    string sName = "NetOut46"
  [NetOut47]
    bool bActive
    bool bEnable = true
    dio dDio = {link=ApplicomIO-1\TOPIC1_A-BLOCKA\%Q47}
    string sID = "NetOut47"
    string sName = "NetOut47"
  [NetOut48]
    bool bActive
    bool bEnable = true
    dio dDio = {link=ApplicomIO-1\TOPIC1_A-BLOCKA\%Q48}
    string sID = "NetOut48"
    string sName = "NetOut48"
  [NetOut49]
    bool bActive
    bool bEnable = true
    dio dDio = {link=ApplicomIO-1\TOPIC1_A-BLOCKA\%Q49}
    string sID = "NetOut49"
    string sName = "NetOut49"
  [NetOut50]
    bool bActive
    bool bEnable = true
    dio dDio = {link=ApplicomIO-1\TOPIC1_A-BLOCKA\%Q50}
    string sID = "NetOut50"
    string sName = "NetOut50"
  [NetOut51]
    bool bActive
    bool bEnable = true
    dio dDio = {link=ApplicomIO-1\TOPIC1_A-BLOCKA\%Q51}
    string sID = "NetOut51"
    string sName = "NetOut51"
  [NetOut52]
    bool bActive
    bool bEnable = true
    dio dDio = {link=ApplicomIO-1\TOPIC1_A-BLOCKA\%Q52}
    string sID = "NetOut52"
    string sName = "NetOut52"
  [NetOut53]
    bool bActive
    bool bEnable = true
    dio dDio = {link=ApplicomIO-1\TOPIC1_A-BLOCKA\%Q53}
    string sID = "NetOut53"
    string sName = "NetOut53"
  [NetOut54]
    bool bActive
    bool bEnable = true
    dio dDio = {link=ApplicomIO-1\TOPIC1_A-BLOCKA\%Q54}
    string sID = "NetOut54"
    string sName = "NetOut54"
  [NetOut55]
    bool bActive
    bool bEnable = true
    dio dDio = {link=ApplicomIO-1\TOPIC1_A-BLOCKA\%Q55}
    string sID = "NetOut55"
    string sName = "NetOut55"
  [NetOut56]
    bool bActive
    bool bEnable = true
    dio dDio = {link=ApplicomIO-1\TOPIC1_A-BLOCKA\%Q56}
    string sID = "NetOut56"
    string sName = "NetOut56"
  [NetOut57]
    bool bActive
    bool bEnable = true
    dio dDio = {link=ApplicomIO-1\TOPIC1_A-BLOCKA\%Q57}
    string sID = "NetOut57"
    string sName = "NetOut57"
  [NetOut58]
    bool bActive
    bool bEnable = true
    dio dDio = {link=ApplicomIO-1\TOPIC1_A-BLOCKA\%Q58}
    string sID = "NetOut58"
    string sName = "NetOut58"
  [NetOut59]
    bool bActive
    bool bEnable = true
    dio dDio = {link=ApplicomIO-1\TOPIC1_A-BLOCKA\%Q59}
    string sID = "NetOut59"
    string sName = "NetOut59"
  [NetOut60]
    bool bActive
    bool bEnable = true
    dio dDio = {link=ApplicomIO-1\TOPIC1_A-BLOCKA\%Q60}
    string sID = "NetOut60"
    string sName = "NetOut60"
  [NetOut61]
    bool bActive
    bool bEnable = true
    dio dDio = {link=ApplicomIO-1\TOPIC1_A-BLOCKA\%Q61}
    string sID = "NetOut61"
    string sName = "NetOut61"
  [NetOut62]
    bool bActive
    bool bEnable = true
    dio dDio = {link=ApplicomIO-1\TOPIC1_A-BLOCKA\%Q62}
    string sID = "NetOut62"
    string sName = "NetOut62"
  [NetOut63]
    bool bActive
    bool bEnable = true
    dio dDio = {link=ApplicomIO-1\TOPIC1_A-BLOCKA\%Q63}
    string sID = "NetOut63"
    string sName = "NetOut63"
  [fOut0]
    bool bActive = true
    bool bEnable = true
    dio dDio = {link=fOut0}
    string sID = "fOut0"
    string sName = "fOut0"
  [valve1]
    bool bActive = true
    bool bEnable = true
    dio dDio = {link=valve1}
    string sID = "valve1"
    string sName = "valve1"
  [valve2]
    bool bActive = true
    bool bEnable = true
    dio dDio = {link=valve2}
    string sID = "valve2"
    string sName = "valve2"
public num nCounter[10]
public string sCondition[6]
  [0] = "!="
  [1] = ">="
  [2] = "> "
  [3] = "< "
  [4] = "<="
  [5] = "=="
public string sOperator[4]
  [0] = "= "
  [1] = "=NUM "
  [2] = "+1"
  [3] = "-1"

--- decompose_num.pgx ---
public program decompose_num(string& x_sItem[] (dimensions=1), string& x_sName (dimensions=1), num& x_nOperator (dimensions=1), num& x_nValue (dimensions=1))
  local num i
  local num l_nPos
  local num l_nSize
  local string l_sItem
  local bool l_bOk
  local string l_sItem2
begin
  //
  // decompose into Index-Operator-Value-Mode
  //
  for i=0 to size(sOperator)-1
    // Operator
    l_nPos=find(x_sItem,sOperator[i])
    if l_nPos!=-1
      x_nOperator=i
      i=size(sOperator)-1
    endIf
  endFor
  if l_nPos!=-1
    // find the Index
    call getSize_num(l_nSize)
    for i=0 to l_nSize-1
      // search it
      call get_num(l_sItem,i)
      if l_sItem==left(x_sItem,l_nPos)
        x_sName=l_sItem
        i=l_nSize-1
      endIf
    endFor
    // get the value
    if x_nOperator==1
      // found the value
      l_sItem2=right(x_sItem,len(x_sItem)-l_nPos-len(sOperator[1]))
      if size(x_sItem)>1
        x_sItem[1]=l_sItem
      endIf
      for i=0 to l_nSize-1
        // search it
        call get_num(l_sItem,i)
        if l_sItem==l_sItem2
          call getValue_num(x_nValue,l_sItem)
          return
        endIf
      endFor
    else
      toNum(right(x_sItem,len(x_sItem)-l_nPos-2),x_nValue,l_bOk)
    endIf
  else
    x_sName=""
  endIf
end

--- decompose_wait.pgx ---
public program decompose_wait(string& x_sItem[] (dimensions=1), string& x_sName (dimensions=1), num& x_nOperator (dimensions=1), num& x_nValue (dimensions=1))
  local num i
  local num l_nPos
  local num l_nSize
  local string l_sItem
  local bool l_bOk
  local string l_sItem2
begin
  //
  // decompose into Index-Operator-Value-Mode
  //
  for i=0 to size(sCondition)-1
    // Operator
    l_nPos=find(x_sItem,sCondition[i])
    if l_nPos!=-1
      x_nOperator=i
      i=size(sCondition)-1
    endIf
  endFor
  if l_nPos!=-1
    // find the Index
    call getSize_num(l_nSize)
    for i=0 to l_nSize-1
      // search it
      call get_num(l_sItem,i)
      if l_sItem==left(x_sItem,l_nPos)
        x_sName=l_sItem
        i=l_nSize-1
      endIf
    endFor
    // get the value
    toNum(right(x_sItem,len(x_sItem)-l_nPos-2),x_nValue,l_bOk)
    if !l_bOk
      // found the value
      l_sItem2=right(x_sItem,len(x_sItem)-l_nPos-len(sCondition[1]))
      if size(x_sItem)>1
        x_sItem[1]=l_sItem
      endIf
      for i=0 to l_nSize-1
        // search it
        call get_num(l_sItem,i)
        if l_sItem==l_sItem2
          call getValue_num(x_nValue,l_sItem)
          return
        endIf
      endFor
    endIf
  else
    x_sName=""
  endIf
end

--- get_num.pgx ---
public program get_num(string& x_sItem[] (dimensions=1), num x_nIndex (dimensions=1))
  local string l_sKey
  local num i
begin
  // OUTPUT
  // start from the first
  l_sKey=first(cCount)
  // search it
  while l_sKey!=""
    x_sItem=l_sKey
    l_sKey=next(cCount[l_sKey])
    if i==x_nIndex
      return
    else
      i=i+1
    endIf
  endWhile
  // start from the first
  l_sKey=first(aCount)
  while l_sKey!=""
    x_sItem=l_sKey
    l_sKey=next(aCount[l_sKey])
    if i==x_nIndex
      return
    else
      i=i+1
    endIf
  endWhile
end

--- getItem_num.pgx ---
public program getItem_num(string& x_sItem (dimensions=1), string x_sId (dimensions=1))
begin
  // get the name
  if isDefined(cCount[x_sId])
    x_sItem=cCount[x_sId].sName
  elseIf isDefined(aCount[x_sId])
    x_sItem=aCount[x_sId].sName
  endIf
end

--- getSize_num.pgx ---
public program getSize_num(num& x_nSize[] (dimensions=1))
begin
  // get the size for the counter
  x_nSize=size(cCount)
  // get the size for the aCounter
  x_nSize=x_nSize+size(aCount)
end

--- getValue_num.pgx ---
public program getValue_num(num& x_nValue[] (dimensions=1), string x_sItem (dimensions=1))
begin
  // Get IT
  if isDefined(cCount[x_sItem])
    x_nValue=cCount[x_sItem].nCount
  elseIf isDefined(aCount[x_sItem])
    x_nValue=aioGet(aCount[x_sItem].aAio)
  else
    // not found
    // toDO
    popUpMsg("value not found: "+x_sItem)
    x_nValue=-1
  endIf
end

--- insert_aCOunt.pgx ---
public program insert_aCount(string x_sItem (dimensions=1), bool x_bActive (dimensions=1), aio x_aDio (dimensions=1))
begin
  // insert a new IO
  if isDefined(aCount[x_sItem])==false and ioStatus(x_aDio)>=0
    insert(aCount[x_sItem])
    aCount[x_sItem].bActive=x_bActive
    aCount[x_sItem].sID=x_sItem
    aCount[x_sItem].sName=x_sItem
    aioLink(aCount[x_sItem].aAio,x_aDio)
    aCount[x_sItem].bEnable=true
  endIf
end

--- insert_aIn.pgx ---
public program insert_aIn(string x_sItem (dimensions=1), bool x_bActive (dimensions=1), aio x_aDio (dimensions=1))
begin
  // insert a new IO
  if isDefined(aInput[x_sItem])==false and ioStatus(x_aDio)>=0
    insert(aInput[x_sItem])
    aInput[x_sItem].bActive=x_bActive
    aInput[x_sItem].sID=x_sItem
    aInput[x_sItem].sName=x_sItem
    aioLink(aInput[x_sItem].aAio,x_aDio)
    aInput[x_sItem].bEnable=true
  endIf
end

--- insert_aOutput.pgx ---
public program insert_aOutput(string x_sItem (dimensions=1), bool x_bActive (dimensions=1), aio x_aDio (dimensions=1))
begin
  // insert a new IO
  if isDefined(aOutput[x_sItem])==false and ioStatus(x_aDio)>=0
    insert(aOutput[x_sItem])
    aOutput[x_sItem].bActive=x_bActive
    aOutput[x_sItem].sID=x_sItem
    aOutput[x_sItem].sName=x_sItem
    aioLink(aOutput[x_sItem].aAio,x_aDio)
    aOutput[x_sItem].bEnable=true
  endIf
end

--- insert_cCount.pgx ---
public program insert_cCount(string x_sItem (dimensions=1), bool x_bActive (dimensions=1), num x_num (dimensions=1))
begin
  // insert a new IO
  if isDefined(cCount[x_sItem])==false
    insert(cCount[x_sItem])
    cCount[x_sItem].bActive=x_bActive
    cCount[x_sItem].sID=x_sItem
    cCount[x_sItem].sName=x_sItem
    cCount[x_sItem].nCount=x_num
    cCount[x_sItem].bEnable=true
  endIf
end

--- insert_dIn.pgx ---
public program insert_dIn(string x_sItem (dimensions=1), bool x_bActive (dimensions=1), dio x_dDio (dimensions=1))
begin
  // insert a new IO
  if isDefined(dInput[x_sItem])==false and ioStatus(x_dDio)>=0
    insert(dInput[x_sItem])
    dInput[x_sItem].bActive=x_bActive
    dInput[x_sItem].sID=x_sItem
    dInput[x_sItem].sName=x_sItem
    dioLink(dInput[x_sItem].dDio,x_dDio)
    dInput[x_sItem].bEnable=true
  endIf
end

--- insert_dOut.pgx ---
public program insert_dOut(string x_sItem (dimensions=1), bool x_bActive (dimensions=1), dio x_dDio (dimensions=1))
begin
  // insert a new IO
  if isDefined(dOutput[x_sItem])==false and ioStatus(x_dDio)>=0
    insert(dOutput[x_sItem])
    dOutput[x_sItem].bActive=x_bActive
    dOutput[x_sItem].sID=x_sItem
    dOutput[x_sItem].sName=x_sItem
    dioLink(dOutput[x_sItem].dDio,x_dDio)
    dOutput[x_sItem].bEnable=true
  endIf
end

--- replaceIO.pgx ---
public program replaceIO(string x_sItem (dimensions=1), string x_sMode (dimensions=1), string& x_sReplace (dimensions=1))
  local num i
  local string l_sItemL
  local string l_sItemR
  local string l_sData[5]
  local num l_nPos
  local num l_nCount
  local num l_nPos2
  local string l_sMode[5]
  local num l_nPos_OR
  local num l_nPos_OUT
  local num l_nPos_AND
  local num l_nPos_IN
  local string l_sId
  local string l_sName
  local num l_nOperator
  local num l_nValue
  local string l_sItem
  local bool l_bOk
  local string l_sItem2
begin
  // init
  x_sReplace=x_sItem
  // go on
  if x_sMode=="IF" or x_sMode=="PULSE"
    if find(x_sItem,"IN ")!=-1
      x_sMode="IN"
    elseIf find(x_sItem,"OUT ")!=-1
      x_sMode="OUT"
    endIf
  endIf
  // scan to find IN or OUT
  // look for all the data
  if x_sMode=="IN" or x_sMode=="OUT"
    l_sItemR=x_sItem
    l_sData=l_sData[1]=l_sData[2]=l_sData[3]=l_sData[4]=""
    while l_nPos!=-1
      // scan all
      l_nPos_AND=l_nPos_IN=l_nPos_OR=l_nPos_OUT=99
      l_sMode[l_nCount]=x_sMode
      l_nPos=find(l_sItemR,">")
      if find(l_sItemR,"AND ")!=-1
        l_nPos_AND=find(l_sItemR,"AND ")+4
      endIf
      if find(l_sItemR,"OR ")!=-1
        l_nPos_OR=find(l_sItemR,"OR ")+3
      endIf
      if find(l_sItemR,"OUT ")!=-1
        l_nPos_OUT=find(l_sItemR,"OUT ")+4
      endIf
      if find(l_sItemR,"IN ")!=-1
        l_nPos_IN=find(l_sItemR,"IN ")+3
      endIf
      // find the nearest
      l_nPos2=min(l_nPos_AND,min(l_nPos_OR,min(l_nPos_IN,min(l_nPos_OUT,90))))
      // check for the mode
      if l_nPos2==l_nPos_OUT
        l_sMode[l_nCount]="OUT"
      elseIf l_nPos2==l_nPos_IN
        l_sMode[l_nCount]="IN"
      endIf
      if l_nPos!=-1
        if find(left(l_sItemR,l_nPos),"EMAP ")==-1
          if l_nPos2==-1 or l_nPos<l_nPos2
            l_sData[l_nCount]=left(l_sItemR,l_nPos)
          else
            l_sData[l_nCount]=right(left(l_sItemR,l_nPos),l_nPos-l_nPos2)
          endIf
        endIf
        l_sItemL=left(l_sItemR,l_nPos)
        l_sItemR=right(l_sItemR,len(l_sItemR)-l_nPos-1)
        // increase
        l_nCount=l_nCount+1
      endIf
    endWhile
    // replace
    for i=0 to 4
      l_sId=l_sData[i]
      switch l_sMode[i]
        case "IN"
          if l_sData[i]!="" and isDefined(dInput[l_sId])
            l_nPos=find(x_sReplace,l_sData[i])
            x_sReplace=replace(x_sReplace,dInput[l_sId].sName,len(l_sData[i]),l_nPos)
          endIf
        break
        case "OUT"
          if l_sData[i]!="" and find(l_sData[i],"EMAP ")==-1 and isDefined(dOutput[l_sId])
            l_nPos=find(x_sReplace,l_sData[i])
            x_sReplace=replace(x_sReplace,dOutput[l_sId].sName,len(l_sData[i]),l_nPos)
          endIf
        break
      endSwitch
    endFor
    //
  elseIf x_sMode=="NUM"
    // replace the num tag
    call decompose_num(x_sItem,l_sName,l_nOperator,l_nValue)
    l_nPos=find(x_sItem,l_sName)
    call getItem_num(l_sItem,l_sName)
    if l_sItem!=""
      x_sReplace=replace(x_sReplace,l_sItem,len(l_sName),l_nPos)
    endIf
  elseIf x_sMode=="WAIT"
    // replace the WAIT tag
    call decompose_wait(x_sItem,l_sName,l_nOperator,l_nValue)
    l_nPos=find(x_sItem,l_sName)
    call getItem_num(l_sItem,l_sName)
    if l_sItem!=""
      x_sReplace=replace(x_sReplace,l_sItem,len(l_sName),l_nPos)
    endIf
    // scan again
    toNum(right(x_sItem,len(x_sItem)-l_nPos-2),l_nValue,l_bOk)
    //    if !l_bOk
    //      // found the value
    //      l_sItem2=right(x_sItem,len(x_sItem)-l_nPos-len(sCondition[1]))
    //      if size(x_sItem)>1
    //        x_sItem[1]=l_sItem
    //      endIf
    //      for i=0 to l_nSize-1
    //        // search it
    //        call get_num(l_sItem,i)
    //        if l_sItem==l_sItem2
    //          l_nPos=find(x_sItem,sCondition[l_nOperator])
    //          call getItem_num(l_sItem,l_sName)
    //          if l_sItem!=""
    //            x_sReplace=replace(x_sReplace,l_sItem,len(l_sName),l_nPos)
    //          endIf
    //        endIf
    //      endFor
    //    endIf
  endIf
end

--- resetAll.pgx ---
public program resetAll()
  local string l_sKey
  local num i
begin
  //
  // init all the IN OUT
  //
  // aCOUNT
  l_sKey=first(aCount)
  while l_sKey!=""
    delete(aCount[l_sKey])
    l_sKey=first(aCount)
  endWhile
  // aINPUT
  l_sKey=first(aInput)
  while l_sKey!=""
    delete(aInput[l_sKey])
    l_sKey=first(aInput)
  endWhile
  // aOUTPUT
  l_sKey=first(aOutput)
  while l_sKey!=""
    delete(aOutput[l_sKey])
    l_sKey=first(aOutput)
  endWhile
  // dINPUT
  l_sKey=first(dInput)
  while l_sKey!=""
    delete(dInput[l_sKey])
    l_sKey=first(dInput)
  endWhile
  // dOUTPUT
  l_sKey=first(dOutput)
  while l_sKey!=""
    delete(dOutput[l_sKey])
    l_sKey=first(dOutput)
  endWhile
  // USER IO
  // DIO
  resize(dInUser,1,1)
  dioLink(dInUser,dNull)
  resize(dOutUser,1,1)
  dioLink(dOutUser,dNull)
  resize(aUser,1,10)
  // AIO
  for i=0 to 9
    aioLink(aUser[i],aNull)
  endFor
  // save it
  libSave()
end

--- setInput.pgx ---
public program setInput(num x_nType)
  local num i
begin
  switch x_nType
    //
    // DIGITAL
    //
    case 0
      if ioStatus(fIn0)>=0
        // CS8C
        bCS8=false
        call insert_dIn("fIn0",true,fIn0)
        call insert_dIn("fIn1",true,fIn1)
        call insert_dIn("usrIn0",true,usrIn0)
        call insert_dIn("usrIn1",true,usrIn1)
      else
        bCS8=true
      endIf
    break
    case 1
      // BIO 1
      call insert_dIn("bIn00",false,bIn0)
      call insert_dIn("bIn01",false,bIn1)
      call insert_dIn("bIn02",false,bIn2)
      call insert_dIn("bIn03",false,bIn3)
      call insert_dIn("bIn04",false,bIn4)
      call insert_dIn("bIn05",false,bIn5)
      call insert_dIn("bIn06",false,bIn6)
      call insert_dIn("bIn07",false,bIn7)
      call insert_dIn("bIn08",false,bIn8)
      call insert_dIn("bIn09",false,bIn9)
      call insert_dIn("bIn10",false,bIn10)
      call insert_dIn("bIn11",false,bIn11)
      call insert_dIn("bIn12",false,bIn12)
      call insert_dIn("bIn13",false,bIn13)
      call insert_dIn("bIn14",false,bIn14)
      call insert_dIn("bIn15",false,bIn15)
    break
    case 2
      if bCS8
        // MIO
        call insert_dIn("mIn00",false,mIn0)
        call insert_dIn("mIn01",false,mIn1)
        call insert_dIn("mIn02",false,mIn2)
        call insert_dIn("mIn03",false,mIn3)
        call insert_dIn("mIn04",false,mIn4)
        call insert_dIn("mIn05",false,mIn5)
        call insert_dIn("mIn06",false,mIn6)
        call insert_dIn("mIn07",false,mIn7)
        call insert_dIn("mIn08",false,mIn8)
        call insert_dIn("mIn09",false,mIn9)
        call insert_dIn("mIn10",false,mIn10)
        call insert_dIn("mIn11",false,mIn11)
        call insert_dIn("mIn12",false,mIn12)
        call insert_dIn("mIn13",false,mIn13)
        call insert_dIn("mIn14",false,mIn14)
        call insert_dIn("mIn15",false,mIn15)
        call insert_dIn("mIn16",false,mIn16)
        call insert_dIn("mIn17",false,mIn17)
        call insert_dIn("mIn18",false,mIn18)
        call insert_dIn("mIn19",false,mIn19)
        call insert_dIn("mIn20",false,mIn20)
        call insert_dIn("mIn21",false,mIn21)
        call insert_dIn("mIn22",false,mIn22)
        call insert_dIn("mIn23",false,mIn23)
        call insert_dIn("mIn24",false,mIn24)
        call insert_dIn("mIn25",false,mIn25)
        call insert_dIn("mIn26",false,mIn26)
        call insert_dIn("mIn27",false,mIn27)
        call insert_dIn("mIn28",false,mIn28)
        call insert_dIn("mIn29",false,mIn29)
        call insert_dIn("mIn30",false,mIn30)
        call insert_dIn("mIn31",false,mIn31)
      else
        // BIO2 - MIO
        call insert_dIn("b2In00",false,b2In0)
        call insert_dIn("b2In01",false,b2In1)
        call insert_dIn("b2In02",false,b2In2)
        call insert_dIn("b2In03",false,b2In3)
        call insert_dIn("b2In04",false,b2In4)
        call insert_dIn("b2In05",false,b2In5)
        call insert_dIn("b2In06",false,b2In6)
        call insert_dIn("b2In07",false,b2In7)
        call insert_dIn("b2In08",false,b2In8)
        call insert_dIn("b2In09",false,b2In9)
        call insert_dIn("b2In10",false,b2In10)
        call insert_dIn("b2In11",false,b2In11)
        call insert_dIn("b2In12",false,b2In12)
        call insert_dIn("b2In13",false,b2In13)
        call insert_dIn("b2In14",false,b2In14)
        call insert_dIn("b2In15",false,b2In15)
      endIf
    break
    case 3
      for i=0 to size(MbIn)-1
        // modbus
        if i<10
          call insert_dIn("MbIn00"+toString("",i),false,MbIn[i])
        elseIf i<100
          call insert_dIn("MbIn0"+toString("",i),false,MbIn[i])
        else
          call insert_dIn("MbIn"+toString("",i),false,MbIn[i])
        endIf
      endFor
    break
    case 4
      // USER
      for i=0 to size(dInUser)-1
        // others
        if i<10
          call insert_dIn("userIn00"+toString("",i),false,dInUser[i])
        elseIf i<100
          call insert_dIn("userIn0"+toString("",i),false,dInUser[i])
        else
          call insert_dIn("userIn"+toString("",i),false,dInUser[i])
        endIf
      endFor
    break
    case 5
      // armIO
      call insert_dIn("remIn0",false,cDin0)
      call insert_dIn("remIn1",false,cDin1)
      call insert_dIn("remIn2",false,cDin2)
      call insert_dIn("remIn3",false,cDin3)
      call insert_dIn("remIn4",false,cDin4)
      call insert_dIn("remIn5",false,cDin5)
      call insert_dIn("remIn6",false,cDin6)
      call insert_dIn("remIn7",false,cDin7)
    break
    //
    case 6
        call insert_dIn("NetIn00",false,NetIn0)
        call insert_dIn("NetIn01",false,NetIn1)
        call insert_dIn("NetIn02",false,NetIn2)
        call insert_dIn("NetIn03",false,NetIn3)
        call insert_dIn("NetIn04",false,NetIn4)
        call insert_dIn("NetIn05",false,NetIn5)
        call insert_dIn("NetIn06",false,NetIn6)
        call insert_dIn("NetIn07",false,NetIn7)
        call insert_dIn("NetIn08",false,NetIn8)
        call insert_dIn("NetIn09",false,NetIn9)
        call insert_dIn("NetIn10",false,NetIn10)
        call insert_dIn("NetIn11",false,NetIn11)
        call insert_dIn("NetIn12",false,NetIn12)
        call insert_dIn("NetIn13",false,NetIn13)
        call insert_dIn("NetIn14",false,NetIn14)
        call insert_dIn("NetIn15",false,NetIn15)
        call insert_dIn("NetIn16",false,NetIn16)
        call insert_dIn("NetIn17",false,NetIn17)
        call insert_dIn("NetIn18",false,NetIn18)
        call insert_dIn("NetIn19",false,NetIn19)
        call insert_dIn("NetIn20",false,NetIn20)
        call insert_dIn("NetIn21",false,NetIn21)
        call insert_dIn("NetIn22",false,NetIn22)
        call insert_dIn("NetIn23",false,NetIn23)
        call insert_dIn("NetIn24",false,NetIn24)
        call insert_dIn("NetIn25",false,NetIn25)
        call insert_dIn("NetIn26",false,NetIn26)
        call insert_dIn("NetIn27",false,NetIn27)
        call insert_dIn("NetIn28",false,NetIn28)
        call insert_dIn("NetIn29",false,NetIn29)
        call insert_dIn("NetIn30",false,NetIn30)
        call insert_dIn("NetIn31",false,NetIn31)
        call insert_dIn("NetIn32",false,NetIn32)
        call insert_dIn("NetIn33",false,NetIn33)
        call insert_dIn("NetIn34",false,NetIn34)
        call insert_dIn("NetIn35",false,NetIn35)
        call insert_dIn("NetIn36",false,NetIn36)
        call insert_dIn("NetIn37",false,NetIn37)
        call insert_dIn("NetIn38",false,NetIn38)
        call insert_dIn("NetIn39",false,NetIn39)
        call insert_dIn("NetIn40",false,NetIn40)
        call insert_dIn("NetIn41",false,NetIn41)
        call insert_dIn("NetIn42",false,NetIn42)
        call insert_dIn("NetIn43",false,NetIn43)
        call insert_dIn("NetIn44",false,NetIn44)
        call insert_dIn("NetIn45",false,NetIn45)
        call insert_dIn("NetIn46",false,NetIn46)
        call insert_dIn("NetIn47",false,NetIn47)
        call insert_dIn("NetIn48",false,NetIn48)
        call insert_dIn("NetIn49",false,NetIn49)
        call insert_dIn("NetIn50",false,NetIn50)
        call insert_dIn("NetIn51",false,NetIn51)
        call insert_dIn("NetIn52",false,NetIn52)
        call insert_dIn("NetIn53",false,NetIn53)
        call insert_dIn("NetIn54",false,NetIn54)
        call insert_dIn("NetIn55",false,NetIn55)
        call insert_dIn("NetIn56",false,NetIn56)
        call insert_dIn("NetIn57",false,NetIn57)
        call insert_dIn("NetIn58",false,NetIn58)
        call insert_dIn("NetIn59",false,NetIn59)
        call insert_dIn("NetIn60",false,NetIn60)
        call insert_dIn("NetIn61",false,NetIn61)
        call insert_dIn("NetIn62",false,NetIn62)
        call insert_dIn("NetIn63",false,NetIn63)
    break
      // ANALOGIC
      //
    case 10
      // default no INPUT
    break
    case 11
      // modbus
      for i=0 to size(MbAnaIn)-1
        call insert_aCount("MbAnaIn"+toString("",i),true,MbAnaIn[i])
      endFor
    break
    case 12
      //
      // USER
      //
    break
    case 13
      // armIO
      call insert_aCount("cArmIn0",true,cAin0)
      call insert_aCount("cArmIn1",true,cAin1)
      call insert_aCount("cArmIn2",true,cAin2)
      call insert_aCount("cArmIn3",true,cAin3)
    break
    case 14
      // others
    break
  endSwitch
end

--- setOutput.pgx ---
public program setOutput(num x_nType)
  local num i
begin
  switch x_nType
    //
    // DIGITAL
    //
    case 0
      // valve 1-2 fastOut
      call insert_dOut("valve1",true,valve1)
      call insert_dOut("valve2",true,valve2)
      if ioStatus(fOut0)>=0
        // CS8C
        bCS8=false
        call insert_dOut("fOut0",true,fOut0)
      else
        bCS8=true
      endIf
    break
    case 1
      // BIO 1
      call insert_dOut("bOut00",false,bOut0)
      call insert_dOut("bOut01",false,bOut1)
      call insert_dOut("bOut02",false,bOut2)
      call insert_dOut("bOut03",false,bOut3)
      call insert_dOut("bOut04",false,bOut4)
      call insert_dOut("bOut05",false,bOut5)
      call insert_dOut("bOut06",false,bOut6)
      call insert_dOut("bOut07",false,bOut7)
      call insert_dOut("bOut08",false,bOut8)
      call insert_dOut("bOut09",false,bOut9)
      call insert_dOut("bOut10",false,bOut10)
      call insert_dOut("bOut11",false,bOut11)
      call insert_dOut("bOut12",false,bOut12)
      call insert_dOut("bOut13",false,bOut13)
      call insert_dOut("bOut14",false,bOut14)
      call insert_dOut("bOut15",false,bOut15)
    break
    case 2
      if bCS8
        // MIO
        call insert_dOut("mOut00",false,mOut0)
        call insert_dOut("mOut01",false,mOut1)
        call insert_dOut("mOut02",false,mOut2)
        call insert_dOut("mOut03",false,mOut3)
        call insert_dOut("mOut04",false,mOut4)
        call insert_dOut("mOut05",false,mOut5)
        call insert_dOut("mOut06",false,mOut6)
        call insert_dOut("mOut07",false,mOut7)
        call insert_dOut("mOut08",false,mOut8)
        call insert_dOut("mOut09",false,mOut9)
        call insert_dOut("mOut10",false,mOut10)
        call insert_dOut("mOut11",false,mOut11)
        call insert_dOut("mOut12",false,mOut12)
        call insert_dOut("mOut13",false,mOut13)
        call insert_dOut("mOut14",false,mOut14)
        call insert_dOut("mOut15",false,mOut15)
        call insert_dOut("mOut16",false,mOut16)
        call insert_dOut("mOut17",false,mOut17)
        call insert_dOut("mOut18",false,mOut18)
        call insert_dOut("mOut19",false,mOut19)
        call insert_dOut("mOut20",false,mOut20)
        call insert_dOut("mOut21",false,mOut21)
        call insert_dOut("mOut22",false,mOut22)
        call insert_dOut("mOut23",false,mOut23)
        call insert_dOut("mOut24",false,mOut24)
        call insert_dOut("mOut25",false,mOut25)
        call insert_dOut("mOut26",false,mOut26)
        call insert_dOut("mOut27",false,mOut27)
        call insert_dOut("mOut28",false,mOut28)
        call insert_dOut("mOut29",false,mOut29)
        call insert_dOut("mOut30",false,mOut30)
        call insert_dOut("mOut31",false,mOut31)
      else
        // BIO2 - MIO
        call insert_dOut("b2Out00",false,b2Out0)
        call insert_dOut("b2Out01",false,b2Out1)
        call insert_dOut("b2Out02",false,b2Out2)
        call insert_dOut("b2Out03",false,b2Out3)
        call insert_dOut("b2Out04",false,b2Out4)
        call insert_dOut("b2Out05",false,b2Out5)
        call insert_dOut("b2Out06",false,b2Out6)
        call insert_dOut("b2Out07",false,b2Out7)
        call insert_dOut("b2Out08",false,b2Out8)
        call insert_dOut("b2Out09",false,b2Out9)
        call insert_dOut("b2Out10",false,b2Out10)
        call insert_dOut("b2Out11",false,b2Out11)
        call insert_dOut("b2Out12",false,b2Out12)
        call insert_dOut("b2Out13",false,b2Out13)
        call insert_dOut("b2Out14",false,b2Out14)
        call insert_dOut("b2Out15",false,b2Out15)
      endIf
    break
    case 3
      for i=0 to size(MbOut)-1
        // modbus
        if i<10
          call insert_dOut("MbOut00"+toString("",i),false,MbOut[i])
        elseIf i<100
          call insert_dOut("MbOut0"+toString("",i),false,MbOut[i])
        else
          call insert_dOut("MbOut"+toString("",i),false,MbOut[i])
        endIf
      endFor
    break
    case 4
      // USER
      for i=0 to size(dOutUser)-1
        // modbus
        if i<10
          call insert_dOut("userOut00"+toString("",i),false,dOutUser[i])
        elseIf i<100
          call insert_dOut("userOut0"+toString("",i),false,dOutUser[i])
        else
          call insert_dOut("userOut"+toString("",i),false,dOutUser[i])
        endIf
      endFor
    break
    case 5
      // armIO
      call insert_dOut("remOut0",false,cDout0)
      call insert_dOut("remOut1",false,cDout1)
      call insert_dOut("remOut2",false,cDout2)
      call insert_dOut("remOut3",false,cDout3)
      call insert_dOut("remOut4",false,cDout4)
      call insert_dOut("remOut5",false,cDout5)
      call insert_dOut("remOut6",false,cDout6)
      call insert_dOut("remOut7",false,cDout7)
    break
    case 6
        call insert_dOut("NetOut00",false,NetOut0)
        call insert_dOut("NetOut01",false,NetOut1)
        call insert_dOut("NetOut02",false,NetOut2)
        call insert_dOut("NetOut03",false,NetOut3)
        call insert_dOut("NetOut04",false,NetOut4)
        call insert_dOut("NetOut05",false,NetOut5)
        call insert_dOut("NetOut06",false,NetOut6)
        call insert_dOut("NetOut07",false,NetOut7)
        call insert_dOut("NetOut08",false,NetOut8)
        call insert_dOut("NetOut09",false,NetOut9)
        call insert_dOut("NetOut10",false,NetOut10)
        call insert_dOut("NetOut11",false,NetOut11)
        call insert_dOut("NetOut12",false,NetOut12)
        call insert_dOut("NetOut13",false,NetOut13)
        call insert_dOut("NetOut14",false,NetOut14)
        call insert_dOut("NetOut15",false,NetOut15)
        call insert_dOut("NetOut16",false,NetOut16)
        call insert_dOut("NetOut17",false,NetOut17)
        call insert_dOut("NetOut18",false,NetOut18)
        call insert_dOut("NetOut19",false,NetOut19)
        call insert_dOut("NetOut20",false,NetOut20)
        call insert_dOut("NetOut21",false,NetOut21)
        call insert_dOut("NetOut22",false,NetOut22)
        call insert_dOut("NetOut23",false,NetOut23)
        call insert_dOut("NetOut24",false,NetOut24)
        call insert_dOut("NetOut25",false,NetOut25)
        call insert_dOut("NetOut26",false,NetOut26)
        call insert_dOut("NetOut27",false,NetOut27)
        call insert_dOut("NetOut28",false,NetOut28)
        call insert_dOut("NetOut29",false,NetOut29)
        call insert_dOut("NetOut30",false,NetOut30)
        call insert_dOut("NetOut31",false,NetOut31)
        call insert_dOut("NetOut32",false,NetOut32)
        call insert_dOut("NetOut33",false,NetOut33)
        call insert_dOut("NetOut34",false,NetOut34)
        call insert_dOut("NetOut35",false,NetOut35)
        call insert_dOut("NetOut36",false,NetOut36)
        call insert_dOut("NetOut37",false,NetOut37)
        call insert_dOut("NetOut38",false,NetOut38)
        call insert_dOut("NetOut39",false,NetOut39)
        call insert_dOut("NetOut40",false,NetOut40)
        call insert_dOut("NetOut41",false,NetOut41)
        call insert_dOut("NetOut42",false,NetOut42)
        call insert_dOut("NetOut43",false,NetOut43)
        call insert_dOut("NetOut44",false,NetOut44)
        call insert_dOut("NetOut45",false,NetOut45)
        call insert_dOut("NetOut46",false,NetOut46)
        call insert_dOut("NetOut47",false,NetOut47)
        call insert_dOut("NetOut48",false,NetOut48)
        call insert_dOut("NetOut49",false,NetOut49)
        call insert_dOut("NetOut50",false,NetOut50)
        call insert_dOut("NetOut51",false,NetOut51)
        call insert_dOut("NetOut52",false,NetOut52)
        call insert_dOut("NetOut53",false,NetOut53)
        call insert_dOut("NetOut54",false,NetOut54)
        call insert_dOut("NetOut55",false,NetOut55)
        call insert_dOut("NetOut56",false,NetOut56)
        call insert_dOut("NetOut57",false,NetOut57)
        call insert_dOut("NetOut58",false,NetOut58)
        call insert_dOut("NetOut59",false,NetOut59)
        call insert_dOut("NetOut60",false,NetOut60)
        call insert_dOut("NetOut61",false,NetOut61)
        call insert_dOut("NetOut62",false,NetOut62)
        call insert_dOut("NetOut63",false,NetOut63)
    break
    //
      // ANALOGIC
      //
    case 10
      // default use the COUNTER
      call insert_cCount("num0",true,nCounter[0])
      call insert_cCount("num1",true,nCounter[1])
      call insert_cCount("num2",true,nCounter[2])
      call insert_cCount("num3",true,nCounter[3])
      call insert_cCount("num4",true,nCounter[4])
      call insert_cCount("num5",true,nCounter[5])
      call insert_cCount("num6",true,nCounter[6])
      call insert_cCount("num7",true,nCounter[7])
      call insert_cCount("num8",true,nCounter[8])
      call insert_cCount("num9",true,nCounter[9])
      // analogic one
      for i=0 to size(aUser)-1
        call insert_aCount("usrNum"+toString("",i),true,aUser[i])
      endFor
    break
    case 11
      // modbus
      for i=0 to size(MbAnaOut)-1
        call insert_aCount("MbAnaOut"+toString("",i),true,MbAnaOut[i])
      endFor
    break
    case 12
      //
      // USER
      //
    break
    case 13
      // armIO
      call insert_aCount("cAout0",true,cAout0)
      call insert_aCount("cAout1",true,cAout1)
      call insert_aCount("cAout2",true,cAout2)
      call insert_aCount("cAout3",true,cAout3)
    break
    case 14
      // others
    break
  endSwitch
end
